// Mitsubishi GX Works2 project: test2   PLC: Q03UDV

PROGRAM MAIN
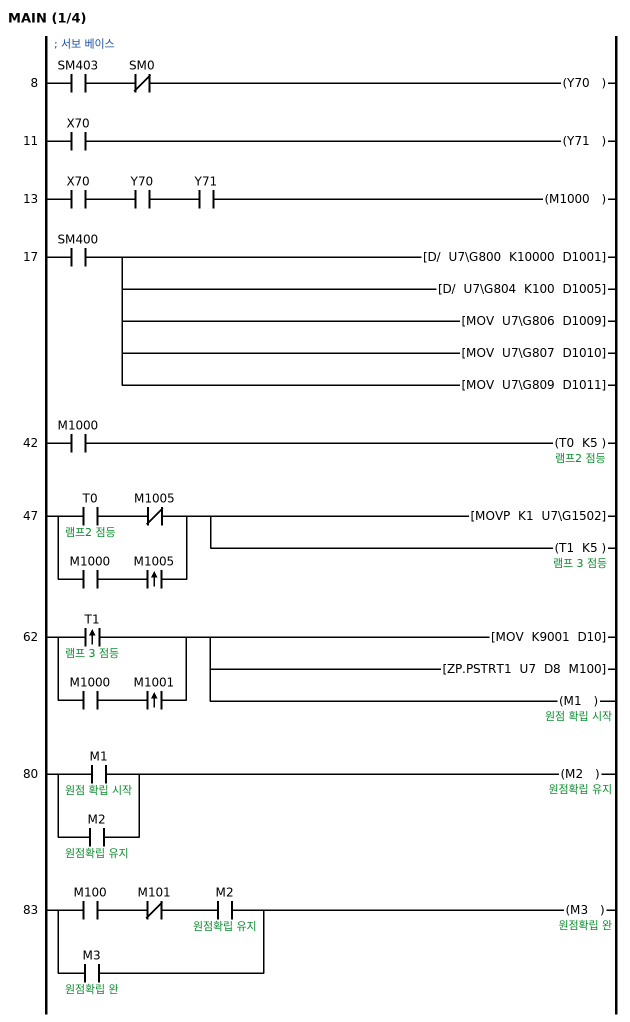
; 서보 베이스
8     LD      SM403
      ANI     SM0
      OUT     Y70
11    LD      X70
      OUT     Y71
13    LD      X70
      AND     Y70
      AND     Y71
      OUT     M1000
17    LD      SM400
      D/      U7\G800 K10000 D1001
      D/      U7\G804 K100 D1005
      MOV     U7\G806 D1009
      MOV     U7\G807 D1010
      MOV     U7\G809 D1011
42    LD      M1000
      OUT     T0 K5  ; 램프2 점등
47    LD      T0  ; 램프2 점등
      ANI     M1005
      LD      M1000
      ANDP    M1005
      ORB
      MOVP    K1 U7\G1502
      OUT     T1 K5  ; 램프 3 점등
62    LDP     T1  ; 램프 3 점등
      LD      M1000
      ANDP    M1001
      ORB
      MOV     K9001 D10
      ZP.PSTRT1 U7 D8 M100
      OUT     M1  ; 원점 확립 시작
80    LD      M1  ; 원점 확립 시작
      OR      M2  ; 원점확립 유지
      OUT     M2  ; 원점확립 유지
83    LD      M100
      ANI     M101
      AND     M2  ; 원점확립 유지
      OR      M3  ; 원점확립 완
      OUT     M3  ; 원점확립 완
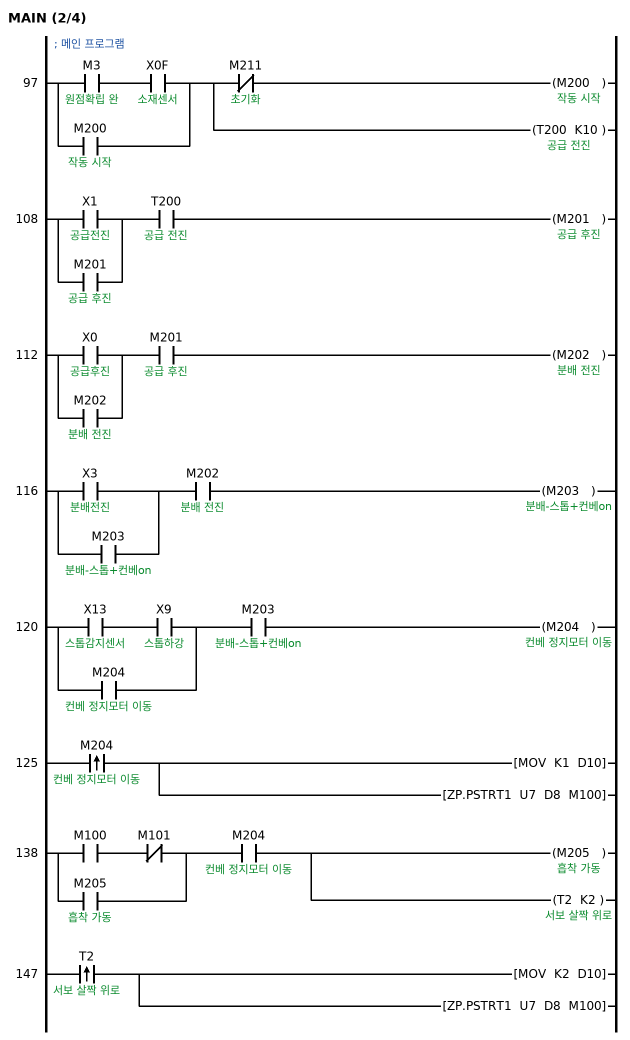
; 메인 프로그램
97    LD      M3  ; 원점확립 완
      AND     X0F  ; 소재센서
      OR      M200  ; 작동 시작
      MPS
      ANI     M211  ; 초기화
      OUT     M200  ; 작동 시작
      MPP
      OUT     T200 K10  ; 공급 전진
108   LD      X1  ; 공급전진
      OR      M201  ; 공급 후진
      AND     T200  ; 공급 전진
      OUT     M201  ; 공급 후진
112   LD      X0  ; 공급후진
      OR      M202  ; 분배 전진
      AND     M201  ; 공급 후진
      OUT     M202  ; 분배 전진
116   LD      X3  ; 분배전진
      OR      M203  ; 분배-스톱+컨베on
      AND     M202  ; 분배 전진
      OUT     M203  ; 분배-스톱+컨베on
120   LD      X13  ; 스톱감지센서
      AND     X9  ; 스톱하강
      OR      M204  ; 컨베 정지모터 이동
      AND     M203  ; 분배-스톱+컨베on
      OUT     M204  ; 컨베 정지모터 이동
125   LDP     M204  ; 컨베 정지모터 이동
      MOV     K1 D10
      ZP.PSTRT1 U7 D8 M100
138   LD      M100
      ANI     M101
      OR      M205  ; 흡착 가동
      AND     M204  ; 컨베 정지모터 이동
      OUT     M205  ; 흡착 가동
      OUT     T2 K2  ; 서보 살짝 위로
147   LDP     T2  ; 서보 살짝 위로
      MOV     K2 D10
      ZP.PSTRT1 U7 D8 M100
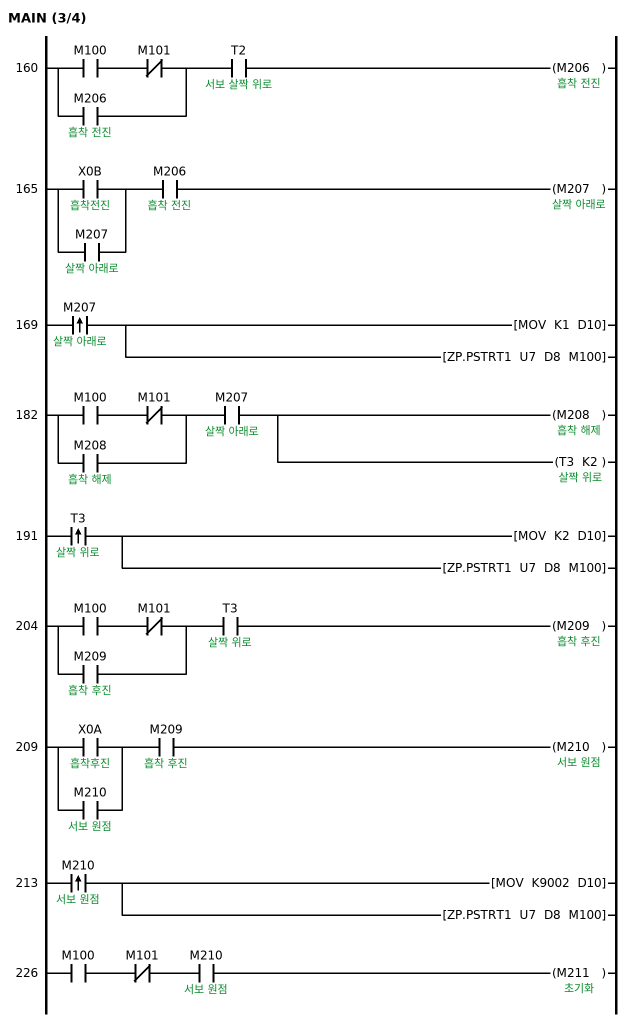
160   LD      M100
      ANI     M101
      OR      M206  ; 흡착 전진
      AND     T2  ; 서보 살짝 위로
      OUT     M206  ; 흡착 전진
165   LD      X0B  ; 흡착전진
      OR      M207  ; 살짝 아래로
      AND     M206  ; 흡착 전진
      OUT     M207  ; 살짝 아래로
169   LDP     M207  ; 살짝 아래로
      MOV     K1 D10
      ZP.PSTRT1 U7 D8 M100
182   LD      M100
      ANI     M101
      OR      M208  ; 흡착 해제
      AND     M207  ; 살짝 아래로
      OUT     M208  ; 흡착 해제
      OUT     T3 K2  ; 살짝 위로
191   LDP     T3  ; 살짝 위로
      MOV     K2 D10
      ZP.PSTRT1 U7 D8 M100
204   LD      M100
      ANI     M101
      OR      M209  ; 흡착 후진
      AND     T3  ; 살짝 위로
      OUT     M209  ; 흡착 후진
209   LD      X0A  ; 흡착후진
      OR      M210  ; 서보 원점
      AND     M209  ; 흡착 후진
      OUT     M210  ; 서보 원점
213   LDP     M210  ; 서보 원점
      MOV     K9002 D10
      ZP.PSTRT1 U7 D8 M100
226   LD      M100
      ANI     M101
      AND     M210  ; 서보 원점
      OUT     M211  ; 초기화
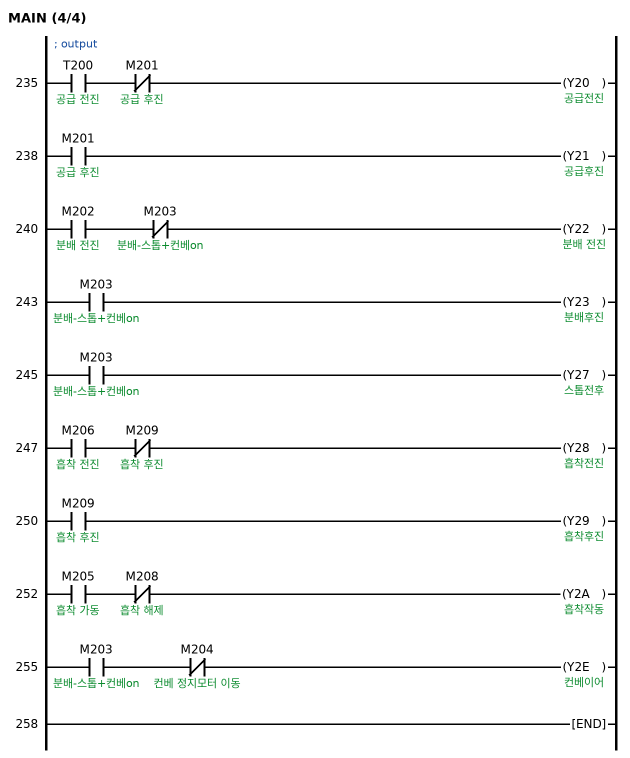
; output
235   LD      T200  ; 공급 전진
      ANI     M201  ; 공급 후진
      OUT     Y20  ; 공급전진
238   LD      M201  ; 공급 후진
      OUT     Y21  ; 공급후진
240   LD      M202  ; 분배 전진
      ANI     M203  ; 분배-스톱+컨베on
      OUT     Y22  ; 분배 전진
243   LD      M203  ; 분배-스톱+컨베on
      OUT     Y23  ; 분배후진
245   LD      M203  ; 분배-스톱+컨베on
      OUT     Y27  ; 스톱전후
247   LD      M206  ; 흡착 전진
      ANI     M209  ; 흡착 후진
      OUT     Y28  ; 흡착전진
250   LD      M209  ; 흡착 후진
      OUT     Y29  ; 흡착후진
252   LD      M205  ; 흡착 가동
      ANI     M208  ; 흡착 해제
      OUT     Y2A  ; 흡착작동
255   LD      M203  ; 분배-스톱+컨베on
      ANI     M204  ; 컨베 정지모터 이동
      OUT     Y2E  ; 컨베이어
258   END
END_PROGRAM

// device comments not shown above
X2  ; 분배후진
X4  ; 가공상승
X5  ; 가공하강
X8  ; 스톱상승
X0C  ; 흡착여부
X11  ; 감지센서
X12  ; 금속센서
X15  ; b1
X16  ; b2
X17  ; b3
X18  ; b4
X19  ; b5
X1A  ; b6
X1B  ; b7
X1C  ; b8
Y24  ; 가공전후
Y2D  ; 드릴
M0  ; 공급전진
M5  ; 분배전진
M6  ; 분배후진
M11  ; 흡착 전진
M12  ; 흡착후진
M13  ; 스톱하강
M14  ; 스톱상승
M15  ; 시퀀스 종료
M18  ; 램프 1 점등
M20  ; 동작조건
M21  ; 동작시작
M22  ; 드릴 시작
M23  ; 가공 하강
M24  ; 가공상승
M25  ; 가공 초기화
M26  ; 공급 후진분배전진
M27  ; 분배후진 컨베이어
M28  ; 감지됨
M29  ; 금속
M30  ; 배출 후진
M31  ; 비금속 종료
M32  ; 시퀀스 종료
M33  ; 시스템 초기화
T4  ; 램프6 점등
T5  ; 램프 7 점등
T6  ; 소등
T20  ; 공급 전진
T21  ; 컨베이어 정지
T22  ; 대기 후 배출 전진
T23  ; 컨베종료금속종료
T24  ; 램2 키고b접점
T25  ; 램2 끄기
T26  ; 램4 키기
T27  ; 램4 끄기
T29  ; 비금속
C20  ; 가공 다음으로
D20  ; 투입 수량
